PROGRAM MAIN
VAR
	Waarde: BYTE;
	nScaledMax: INT := 10;
	potentiometer: INT;
END_VAR

(*
Declareer een variabele van het type INT, met de naam nScaledMax en een initial value van 10. Gebruik hiervoor de Auto Declare functie (zie afbeelding). 
Vervolgens schrijf je de code om de potentiometer-waarde te verschalen naar een getal tussen 0 en nScaledMax.
*)

Waarde:=LREAL_TO_BYTE(nScaledMax*(potentiometer/32767.0));

END_PROGRAM

(* stored: Version 1.1.0.1, ProductVersion 3.1.4024.12
   POU MAIN: Id {674d2829-09d5-468e-a4ba-90184b9a8337}, SpecialFunc None *)
